FUNCTION_BLOCK EjectionGate IMPLEMENTS MachineModule
VAR
	bEnable			: BOOL;
	bDisable        : BOOL;
	bError          : BOOL;
	bOverride       : BOOL;
	bSimulation     : BOOL;
	bStart          : BOOL;
	bStop           : BOOL;
END_VAR

// This is the core module needed that we are creating for our STS and contains everything related to the STS

// To be added
(*
FEEDER

SAT

VBT

EJECT

GATE

SBT

*)

METHOD Disable : BOOL
VAR_INPUT
END_VAR
bEnable:=FALSE;
END_METHOD

METHOD Enable : BOOL
VAR_INPUT
END_VAR
bEnable:=TRUE;
bDisable:=False;
END_METHOD

METHOD Error : BOOL
VAR_INPUT
END_VAR
bEnable:=FALSE;
END_METHOD

METHOD Override : BOOL
VAR_INPUT
END_VAR
END_METHOD

METHOD Reset : BOOL
VAR_INPUT
END_VAR
END_METHOD

METHOD Start : BOOL
VAR_INPUT
END_VAR
END_METHOD

METHOD PUBLIC StateMachine
VAR_INPUT
END_VAR
END_METHOD

METHOD Stop : BOOL
VAR_INPUT
END_VAR
END_METHOD

END_FUNCTION_BLOCK

(* stored: Version 1.1.0.1, ProductVersion 3.1.4024.12
   POU EjectionGate: Id {da28725f-c96c-4149-b087-60e361176424}, SpecialFunc None
   Method Disable: Id {30f9b8a1-fce6-48d7-a259-36e2cfdd0e0a}
   Method Enable: Id {c8d000f4-193e-4fa6-a733-11f5e48ad0fd}
   Method Error: Id {2aabecdd-e1c0-4a1a-8bde-b8d8832784f9}
   Method Override: Id {d3433c37-471c-4059-a5e9-093e7b9dbe69}
   Method Reset: Id {e5968cc0-0142-4d07-8ec1-555714f14f73}
   Method Start: Id {28cad696-c7b9-4fd9-baa1-70b346ed0d77}
   Method StateMachine: Id {2967c8e0-1a88-47c6-85bb-06a288e4b591}
   Method Stop: Id {ce3ad334-fff8-4810-9c73-ab75a82d93bf} *)
